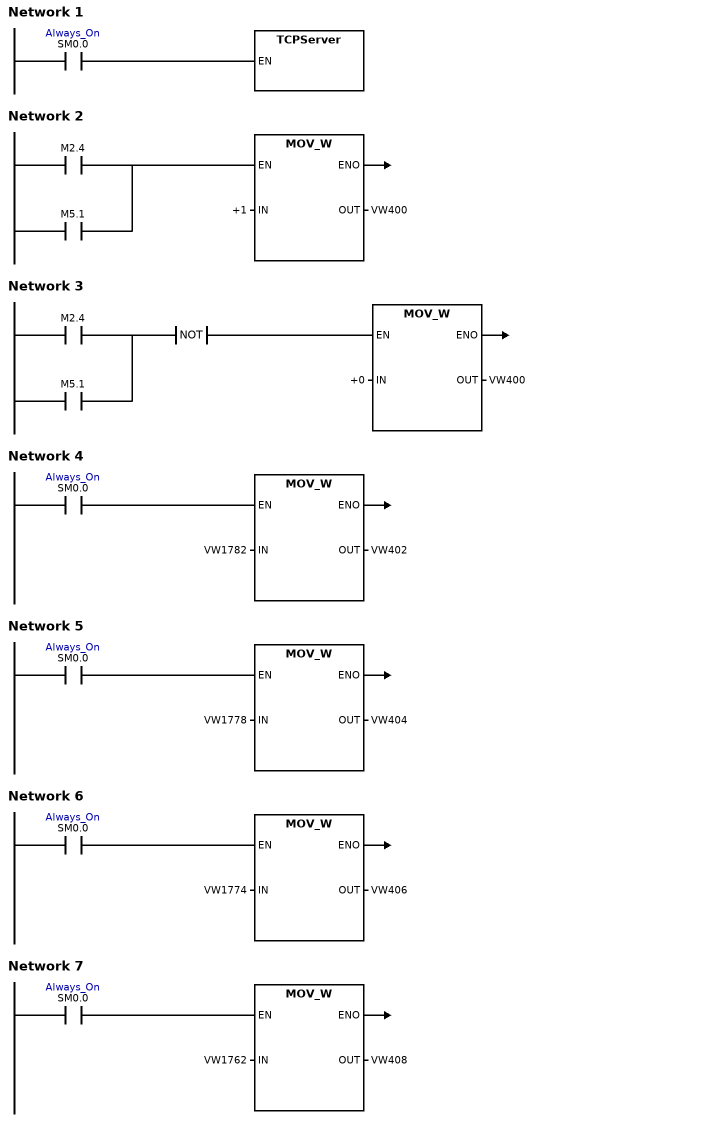
[picture p24: SBR8 networks 1-7]
Network 1
LD     Always_On:SM0.0
CALL   TCPServer:SBR10
Network 2
LD     M2.4
O      M5.1
MOVW   +1, VW400
Network 3
LD     M2.4
O      M5.1
NOT
MOVW   +0, VW400
Network 4
LD     Always_On:SM0.0
MOVW   VW1782, VW402
Network 5
LD     Always_On:SM0.0
MOVW   VW1778, VW404
Network 6
LD     Always_On:SM0.0
MOVW   VW1774, VW406
Network 7
LD     Always_On:SM0.0
MOVW   VW1762, VW408
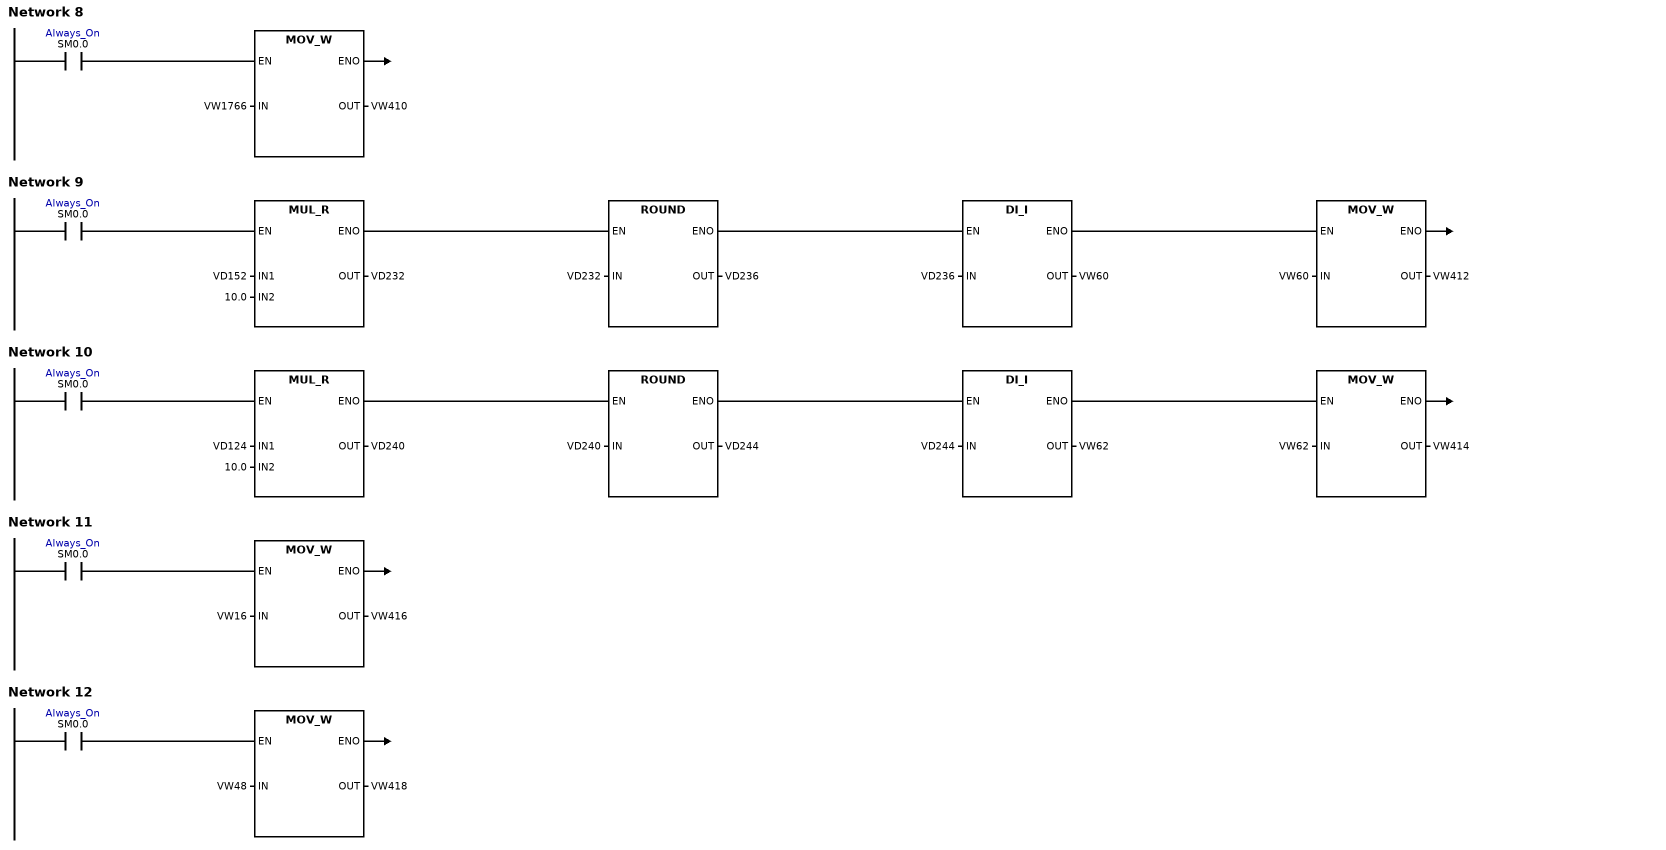
Network 8
LD     Always_On:SM0.0
MOVW   VW1766, VW410
Network 9
LD     Always_On:SM0.0
MOVR   VD152, VD232
AENO
*R     10.0, VD232
AENO
ROUND  VD232, VD236
AENO
DTI    VD236, VW60
AENO
MOVW   VW60, VW412
Network 10
LD     Always_On:SM0.0
MOVR   VD124, VD240
AENO
*R     10.0, VD240
AENO
ROUND  VD240, VD244
AENO
DTI    VD244, VW62
AENO
MOVW   VW62, VW414
Network 11
LD     Always_On:SM0.0
MOVW   VW16, VW416
Network 12
LD     Always_On:SM0.0
MOVW   VW48, VW418
END_SUBROUTINE_BLOCK

// SBR9: protected block, not included

SUBROUTINE_BLOCK TCPServer:SBR10
TITLE=
BEGIN
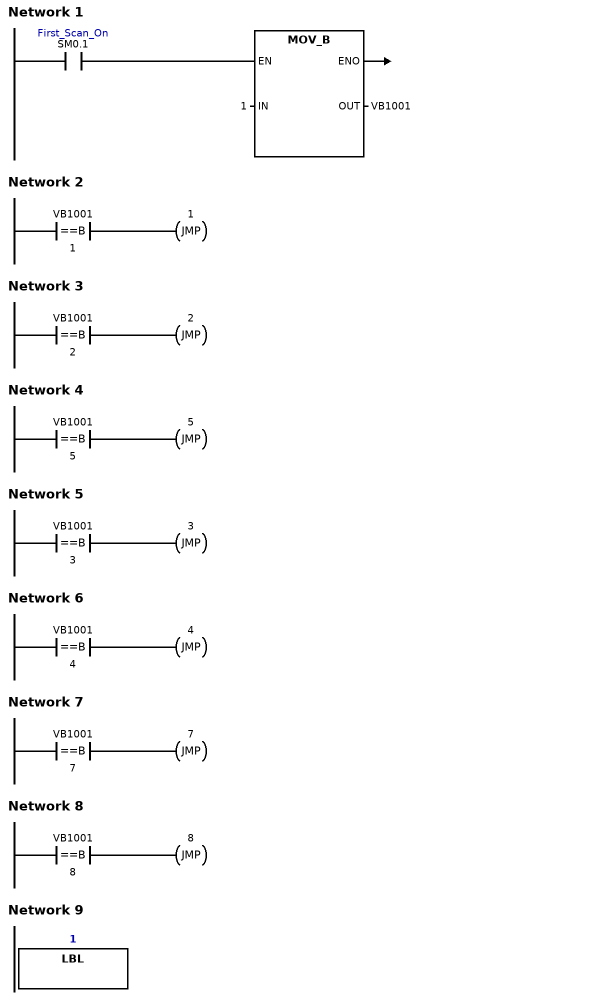
Network 1
LD     First_Scan_On:SM0.1
MOVB   1, VB1001
Network 2
LDB=   VB1001, 1
JMP    1
Network 3
LDB=   VB1001, 2
JMP    2
Network 4
LDB=   VB1001, 5
JMP    5
Network 5
LDB=   VB1001, 3
JMP    3
Network 6
LDB=   VB1001, 4
JMP    4
Network 7
LDB=   VB1001, 7
JMP    7
Network 8
LDB=   VB1001, 8
JMP    8
Network 9
LBL    1
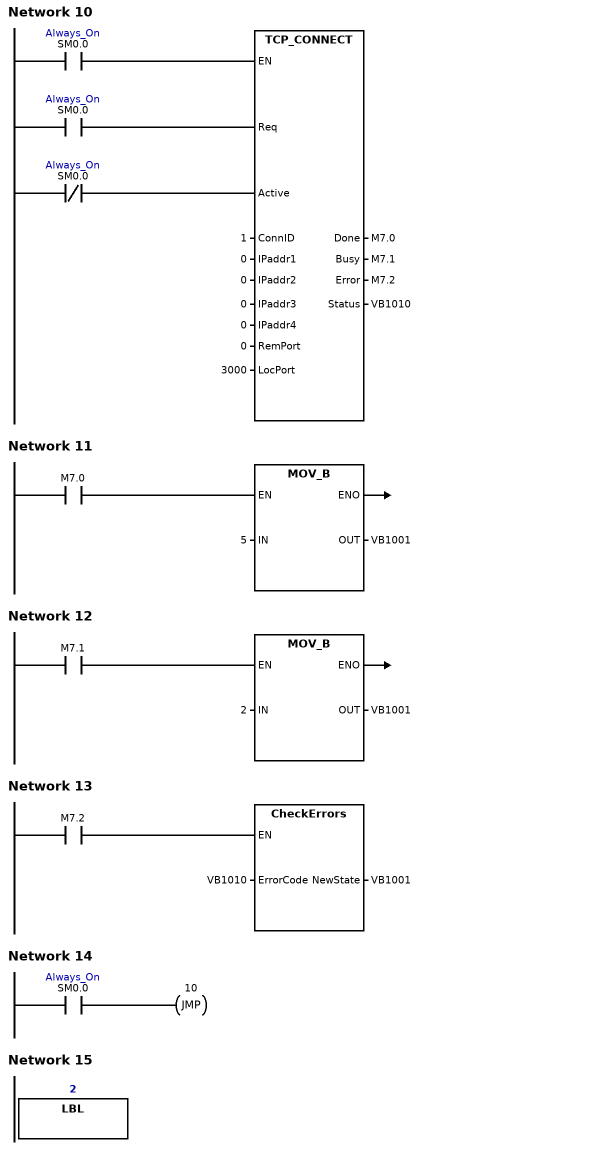
Network 10
LD     Always_On:SM0.0
=      L60.0
LD     Always_On:SM0.0
=      L63.7
LDN    Always_On:SM0.0
=      L63.6
LD     L60.0
CALL   TCP_CONNECT:SBR9, L63.7, L63.6, 1, 0, 0, 0, 0, 0, 3000, M7.0, M7.1, M7.2, VB1010
Network 11
LD     M7.0
MOVB   5, VB1001
Network 12
LD     M7.1
MOVB   2, VB1001
Network 13
LD     M7.2
CALL   CheckErrors:SBR15, VB1010, VB1001
Network 14
LD     Always_On:SM0.0
JMP    10
Network 15
LBL    2
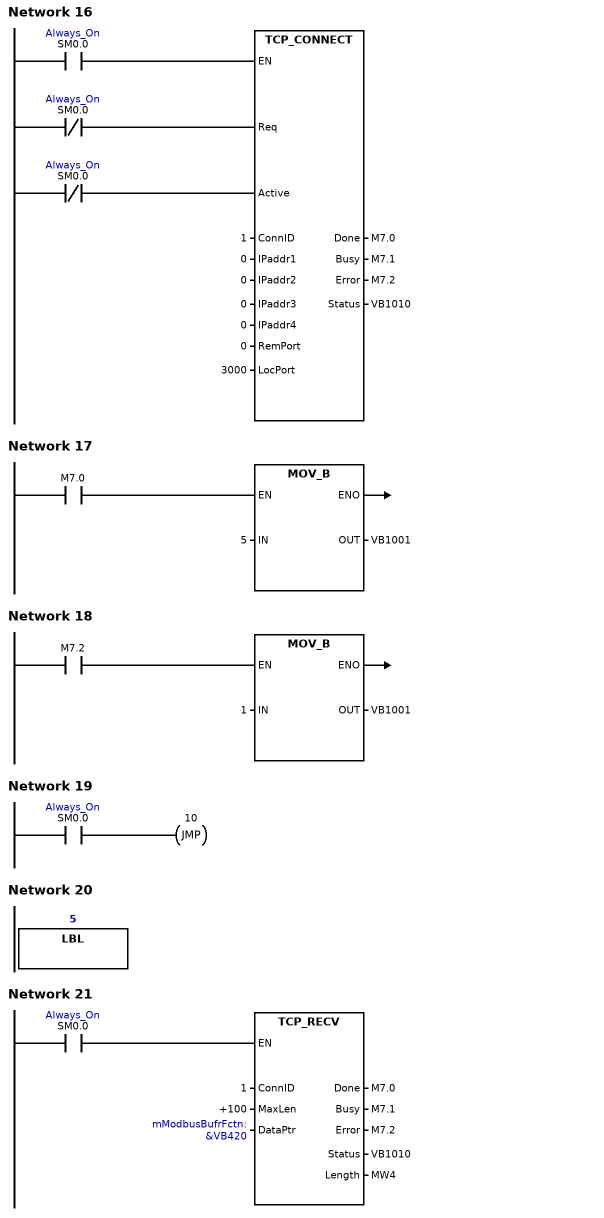
Network 16
LD     Always_On:SM0.0
=      L60.0
LDN    Always_On:SM0.0
=      L63.7
LDN    Always_On:SM0.0
=      L63.6
LD     L60.0
CALL   TCP_CONNECT:SBR9, L63.7, L63.6, 1, 0, 0, 0, 0, 0, 3000, M7.0, M7.1, M7.2, VB1010
Network 17
LD     M7.0
MOVB   5, VB1001
Network 18
LD     M7.2
MOVB   1, VB1001
Network 19
LD     Always_On:SM0.0
JMP    10
Network 20
LBL    5
Network 21
LD     Always_On:SM0.0
CALL   TCP_RECV:SBR11, 1, +100, &mModbusBufrFctn:VB420, M7.0, M7.1, M7.2, VB1010, MW4
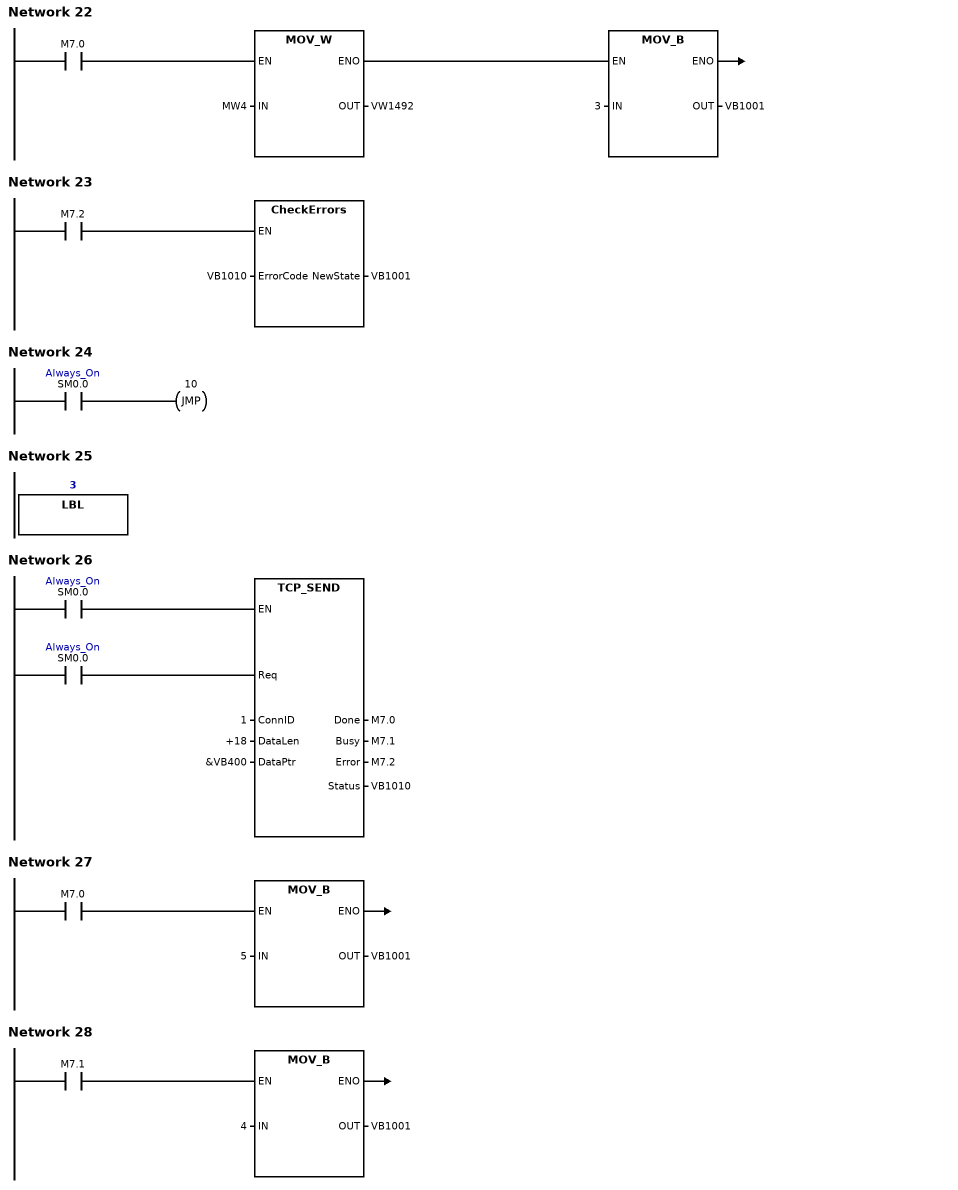
Network 22
LD     M7.0
MOVW   MW4, VW1492
AENO
MOVB   3, VB1001
Network 23
LD     M7.2
CALL   CheckErrors:SBR15, VB1010, VB1001
Network 24
LD     Always_On:SM0.0
JMP    10
Network 25
LBL    3
Network 26
LD     Always_On:SM0.0
=      L60.0
LD     Always_On:SM0.0
=      L63.7
LD     L60.0
CALL   TCP_SEND:SBR12, L63.7, 1, +18, &VB400, M7.0, M7.1, M7.2, VB1010
Network 27
LD     M7.0
MOVB   5, VB1001
Network 28
LD     M7.1
MOVB   4, VB1001
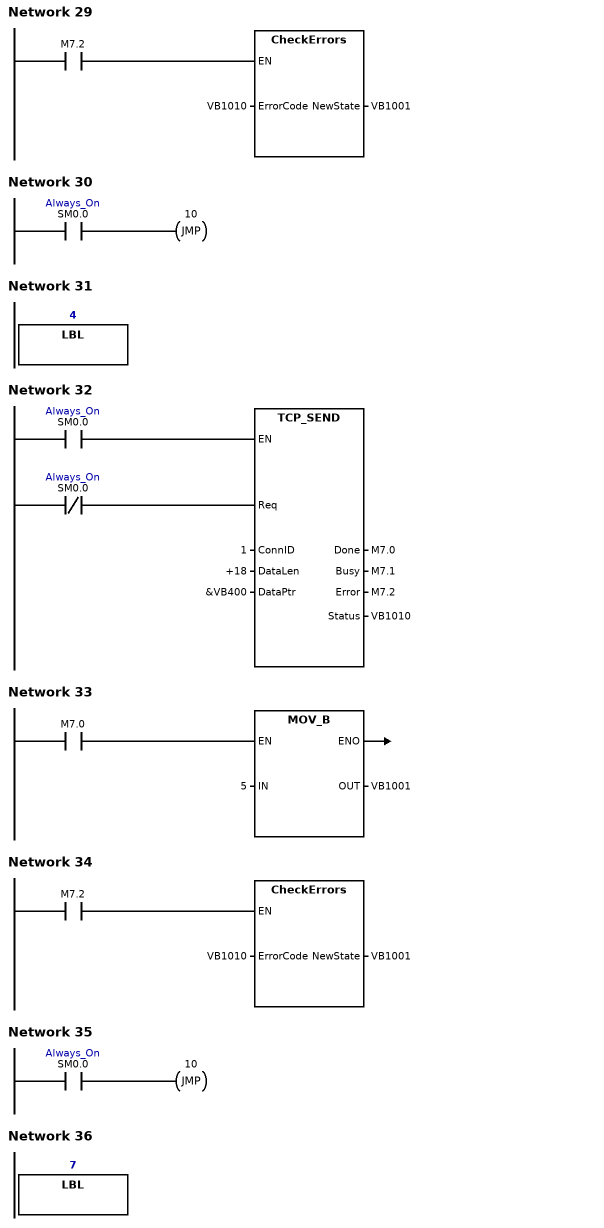
Network 29
LD     M7.2
CALL   CheckErrors:SBR15, VB1010, VB1001
Network 30
LD     Always_On:SM0.0
JMP    10
Network 31
LBL    4
Network 32
LD     Always_On:SM0.0
=      L60.0
LDN    Always_On:SM0.0
=      L63.7
LD     L60.0
CALL   TCP_SEND:SBR12, L63.7, 1, +18, &VB400, M7.0, M7.1, M7.2, VB1010
Network 33
LD     M7.0
MOVB   5, VB1001
Network 34
LD     M7.2
CALL   CheckErrors:SBR15, VB1010, VB1001
Network 35
LD     Always_On:SM0.0
JMP    10
Network 36
LBL    7
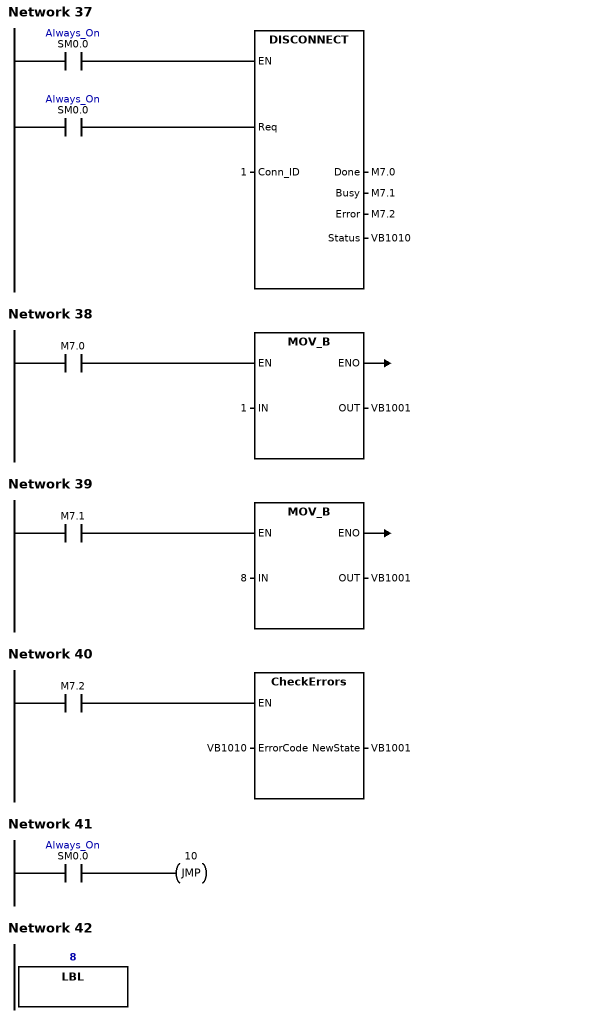
Network 37
LD     Always_On:SM0.0
=      L60.0
LD     Always_On:SM0.0
=      L63.7
LD     L60.0
CALL   DISCONNECT:SBR13, L63.7, 1, M7.0, M7.1, M7.2, VB1010
Network 38
LD     M7.0
MOVB   1, VB1001
Network 39
LD     M7.1
MOVB   8, VB1001
Network 40
LD     M7.2
CALL   CheckErrors:SBR15, VB1010, VB1001
Network 41
LD     Always_On:SM0.0
JMP    10
Network 42
LBL    8
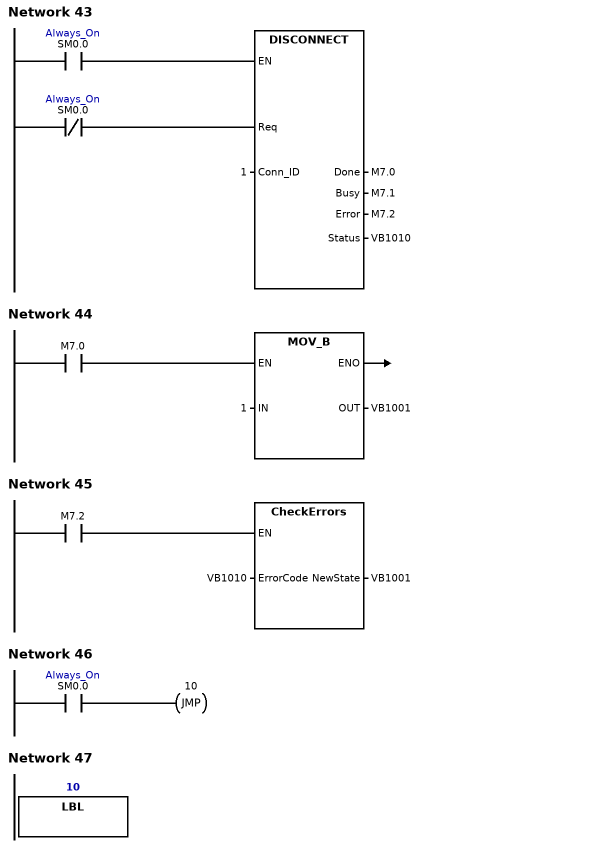
Network 43
LD     Always_On:SM0.0
=      L60.0
LDN    Always_On:SM0.0
=      L63.7
LD     L60.0
CALL   DISCONNECT:SBR13, L63.7, 1, M7.0, M7.1, M7.2, VB1010
Network 44
LD     M7.0
MOVB   1, VB1001
Network 45
LD     M7.2
CALL   CheckErrors:SBR15, VB1010, VB1001
Network 46
LD     Always_On:SM0.0
JMP    10
Network 47
LBL    10
END_SUBROUTINE_BLOCK

// SBR11: protected block, not included

// SBR12: protected block, not included

// SBR13: protected block, not included

// SBR14: protected block, not included

SUBROUTINE_BLOCK CheckErrors:SBR15
TITLE=
VAR_INPUT
ErrorCode:BYTE;	// LB0 
END_VAR
VAR_OUTPUT
NewState:BYTE;	// LB1 
END_VAR
BEGIN
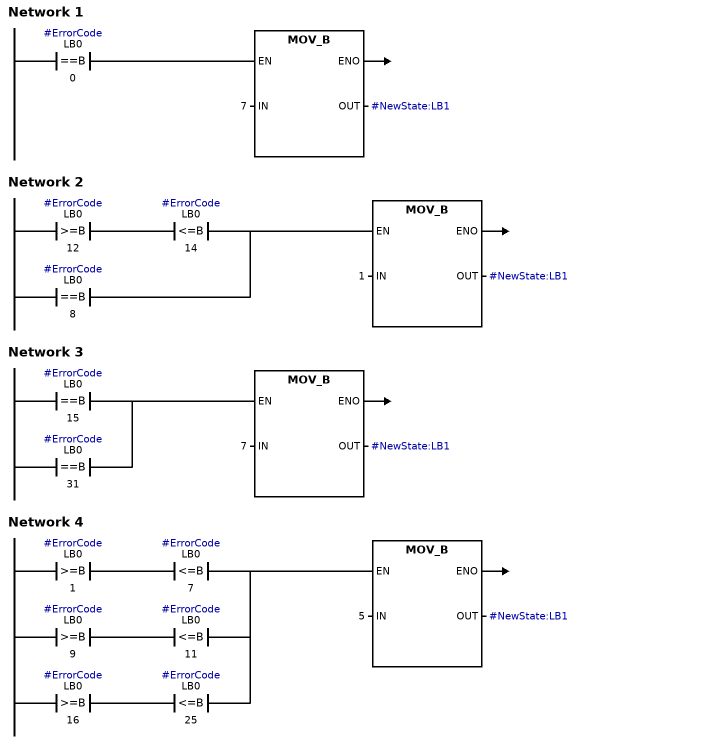
Network 1
LDB=   #ErrorCode:LB0, 0
MOVB   7, #NewState:LB1
Network 2
LDB>=  #ErrorCode:LB0, 12
AB<=   #ErrorCode:LB0, 14
OB=    #ErrorCode:LB0, 8
MOVB   1, #NewState:LB1
Network 3
LDB=   #ErrorCode:LB0, 15
OB=    #ErrorCode:LB0, 31
MOVB   7, #NewState:LB1
Network 4
LDB>=  #ErrorCode:LB0, 1
AB<=   #ErrorCode:LB0, 7
LDB>=  #ErrorCode:LB0, 9
AB<=   #ErrorCode:LB0, 11
OLD
LDB>=  #ErrorCode:LB0, 16
AB<=   #ErrorCode:LB0, 25
OLD
MOVB   5, #NewState:LB1
END_SUBROUTINE_BLOCK

// INT1: protected block, not included

DATA_BLOCK_TAB _PLC_DATA_1
BEGIN
VB1      16#5
VB3      16#1E
VB5      16#3C
VB7      16#1E
VB25     16#8
VB27     16#5
VB33     16#3
VB102    16#18
VB103    16#6A
VB104    16#42
VB105    16#7A
VB106    16#0
VB107    16#0
VB108    16#42
VB109    16#80
VB112    16#42
VB113    16#9A
VB116    16#C3
VB117    16#D7
VB124    16#C3
VB125    16#F1
VB126    16#F
VB130    16#3D
VB131    16#C8
VB132    16#43
VB133    16#1E
VB134    16#28
VB135    16#F6
VB140    16#43
VB141    16#8A
VB142    16#33
VB148    16#42
VB149    16#C8
VB152    16#42
VB153    16#64
VB154    16#E2
VB155    16#BC
VB156    16#C3
VB157    16#C8
VB160    16#42
VB161    16#5C
VB164    16#C3
VB165    16#C8
VB168    16#42
VB169    16#5C
VB204    16#45
VB205    16#C3
VB206    16#50
VB208    16#46
VB209    16#77
VB210    16#20
END_DATA_BLOCK_TAB

DATA_BLOCK_TAB _PLC_DATA_2
BEGIN
VB21     16#0
VB23     16#A
VB143    16#33
VB188    16#BE
VB189    16#E1
VB190    16#FE
VB191    16#0
VB192    16#BE
VB193    16#61
VB194    16#FE
VB195    16#0
VB199    16#0
VB200    16#42
VB201    16#5E
VB212    16#42
VB213    16#64
VB214    16#E2
VB215    16#BC
VB216    16#C3
VB217    16#EF
VB218    16#6E
END_DATA_BLOCK_TAB

DATA_BLOCK_TAB _PLC_DATA_3
BEGIN
VB219    16#8C
END_DATA_BLOCK_TAB

DATA_BLOCK_TAB _PLC_DATA_4
BEGIN
VB37     16#0
VB41     16#0
VB127    16#84
END_DATA_BLOCK_TAB

DATA_BLOCK_TAB _PLC_DATA_5
BEGIN
VB9      16#5
VB11     16#1E
VB43     16#A
VB172    16#C3
VB173    16#C8
VB176    16#42
VB177    16#5C
VB180    16#C3
VB181    16#C8
VB220    16#42
VB221    16#48
END_DATA_BLOCK_TAB

DATA_BLOCK_TAB _PLC_DATA_6
BEGIN
VB45     16#0
VB47     16#0
VB224    16#C3
VB225    16#AF
END_DATA_BLOCK_TAB

DATA_BLOCK_TAB _PLC_DATA_7
BEGIN
VB114    16#66
VB115    16#66
END_DATA_BLOCK_TAB

DATA_BLOCK_TAB _PLC_DATA_8
BEGIN
VB13     16#B4
VB15     16#1E
VB49     16#5
VB51     16#D
VB53     16#A
VB55     16#2
VB57     16#A
VB59     16#2
VB184    16#42
VB185    16#5C
VB228    16#C3
VB229    16#C8
END_DATA_BLOCK_TAB

DATA_BLOCK_TAB _PLC_DATA_9
BEGIN
VB39     16#0
END_DATA_BLOCK_TAB

DATA_BLOCK_TAB _PLC_DATA_10
BEGIN
VB226    16#0
END_DATA_BLOCK_TAB

DATA_BLOCK_TAB _PLC_DATA_11
BEGIN
VB60     16#2
VB61     16#3C
VB62     16#ED
VB63     16#2B
VB232    16#44
VB233    16#F
VB234    16#D
VB235    16#B6
VB238    16#2
VB239    16#3C
VB240    16#C5
VB241    16#96
VB242    16#A9
VB243    16#B2
VB245    16#FF
VB246    16#ED
VB247    16#2B
VB401    16#0
VB403    16#1
VB405    16#1
VB407    16#0
VB409    16#0
VB411    16#0
VB412    16#2
VB413    16#3C
VB414    16#ED
VB415    16#2B
VB800    16#0
VB801    16#1
VB802    16#1
VB803    16#0
VB804    16#0
VB805    16#25
VB807    16#7
VB1000   16#2
VB1001   16#2
VB1003   16#1
VB1004   16#F6
VB1010   16#0
VB1011   16#8
VB1013   16#1
VB1014   16#90
VB1016   16#9
VB1018   16#1C
VB1019   16#D5
VB1035   16#1C
VB1036   16#D6
VB1052   16#1C
VB1053   16#D7
VB1069   16#1C
VB1070   16#D8
VB1086   16#1C
VB1087   16#D9
VB1103   16#1C
VB1104   16#DA
VB1120   16#1C
VB1121   16#DB
VB1136   16#8
VB1138   16#3
VB1139   16#E8
VB1140   16#90
VB1141   16#CD
VB1142   16#A7
VB1143   16#3D
VB1144   16#8
VB1146   16#3
VB1147   16#E9
VB1148   16#8
VB1150   16#3
VB1151   16#EB
VB1152   16#8
VB1154   16#3
VB1155   16#ED
VB1156   16#8
VB1158   16#3
VB1159   16#EF
VB1160   16#40
VB1162   16#1C
VB1163   16#D4
VB1166   16#8
VB1168   16#4
VB1169   16#A0
VB1171   16#1
VB1172   16#F6
VB1185   16#23
VB1189   16#3
VB1190   16#1
VB1191   16#83
VB1192   16#2
VB1195   16#28
VB1437   16#1
VB1442   16#2
VB1761   16#0
VB1763   16#0
VB1765   16#0
VB1767   16#0
VB1769   16#25
VB1771   16#19
VB1773   16#0
VB1775   16#0
VB1777   16#1
VB1779   16#1
VB1781   16#1
VB1783   16#1
END_DATA_BLOCK_TAB

DATA_BLOCK_TAB _PLC_DATA_12
BEGIN
oucTable:VB348 16#40
VB351    16#1
oucConnType:VB352 16#B
oucUdpAddress2:VB359 16#B
oucUdpAddress3:VB360 16#B8
END_DATA_BLOCK_TAB

DATA_BLOCK_TAB _PLC_DATA_13
BEGIN
VB244    16#FF
mModbusBufrSlave:VB419 16#5
VB2886   16#5
END_DATA_BLOCK_TAB

DATA_BLOCK_TAB _PLC_DATA_14
BEGIN
mConnectionTable:VB2674 16#1
VB2675   16#1C
VB2676   16#D4
VB2677   16#9
VB2678   16#C4
VB2679   16#1
VB2682   16#38
VB2684   16#32
VB2685   16#8
VB2687   16#1
VB2688   16#90
VB2690   16#0
VB2692   16#1C
VB2693   16#D5
VB2709   16#1C
VB2710   16#D6
VB2726   16#1C
VB2727   16#D7
VB2743   16#1C
VB2744   16#D8
VB2760   16#1C
VB2761   16#D9
VB2777   16#1C
VB2778   16#DA
VB2794   16#1C
VB2795   16#DB
VB2810   16#8
VB2812   16#A
VB2813   16#72
VB2814   16#90
VB2815   16#CD
VB2816   16#A7
VB2817   16#3D
VB2818   16#8
VB2820   16#A
VB2821   16#73
VB2822   16#8
VB2824   16#A
VB2825   16#75
VB2826   16#8
VB2828   16#A
VB2829   16#77
VB2830   16#8
VB2832   16#A
VB2833   16#79
mOUCTbl:VB2834 16#40
VB2836   16#1C
VB2837   16#D4
VB2840   16#0
VB2842   16#0
VB2843   16#0
VB2845   16#9
VB2846   16#C4
VB2859   16#77
VB2863   16#4F
VB2864   16#1
mMsgBuf_FunctionCode:VB2865 16#3
mMsgBuf_ByteCountRespon:VB2866 16#4C
VB2868   16#1
mMsgBuf_ByteCountReq:VB2870 16#1
VB2872   16#1
VB2874   16#0
VB2876   16#0
VB2878   16#0
VB2879   16#2
VB2880   16#45
VB2881   16#F0
VB2882   16#59
VB3111   16#0
mState:VB3116 16#1
END_DATA_BLOCK_TAB

DATA_BLOCK_TAB _PLC_DATA_15
BEGIN
mOUCTbl_ConnectionType:VB2838 16#B
END_DATA_BLOCK_TAB

DATA_BLOCK_TAB _PLC_DATA_16
BEGIN
VB17     16#0
VB31     16#0
VB35     16#0
VB417    16#0
VB2884   16#0
END_DATA_BLOCK_TAB

DATA_BLOCK_TAB _PLC_DATA_17
BEGIN
VB19     16#0
VB29     16#13
END_DATA_BLOCK_TAB

DATA_BLOCK_TAB _PLC_DATA_19
BEGIN
VB248    16#C3
VB249    16#FA
END_DATA_BLOCK_TAB
